{attribute 'qualified_only'}
{attribute 'strict'}
TYPE eUSVSaveMode :
(
	eSaveWhenPowerfail := 0,
	eSaveEventBased := 1,
	eSaveOnBoth := 2
);
END_TYPE

(* stored: Version 1.1.0.1, ProductVersion 3.1.4024.9
   DUT eUSVSaveMode: Id {4a9a3b1d-9c95-4237-9a84-02637ec5c244} *)
